SUBAPPLICATION ButtonFunc (* Subapplication Type *)
  (* Standard: 61499-2 *)
  (* Version 1.0, 2023-02-19, franz *)
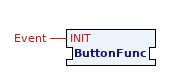
  EVENT_INPUT
    INIT;
  END_EVENT
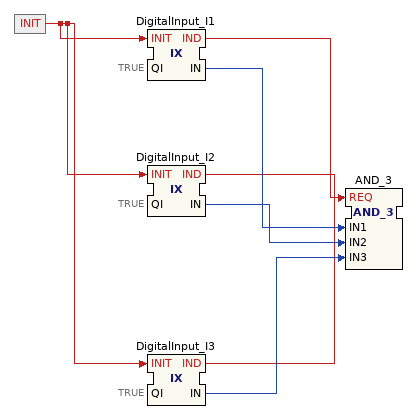
  FBS
    DigitalInput_I1 : IX(QI := TRUE);
    DigitalInput_I2 : IX(QI := TRUE);
    DigitalInput_I3 : IX(QI := TRUE);
    AND_3 : AND_3;
  END_FBS
  EVENT_CONNECTIONS
    INIT TO DigitalInput_I1.INIT;
    INIT TO DigitalInput_I2.INIT;
    INIT TO DigitalInput_I3.INIT;
    DigitalInput_I1.IND TO AND_3.REQ;
    DigitalInput_I2.IND TO AND_3.REQ;
    DigitalInput_I3.IND TO AND_3.REQ;
  END_CONNECTIONS
  DATA_CONNECTIONS
    DigitalInput_I1.IN TO AND_3.IN1;
    DigitalInput_I2.IN TO AND_3.IN2;
    DigitalInput_I3.IN TO AND_3.IN3;
  END_CONNECTIONS
END_SUBAPPLICATION
